// TIA Portal V19 export
FUNCTION "CallSettings" : Void   // FC8, LAD
// Call of settings blocks
// stored: IsIECCheckEnabled true, SetENOAutomatically false
BEGIN

REGION Network 1: Set set PLC date and time
   // Change local date and time of the PLC
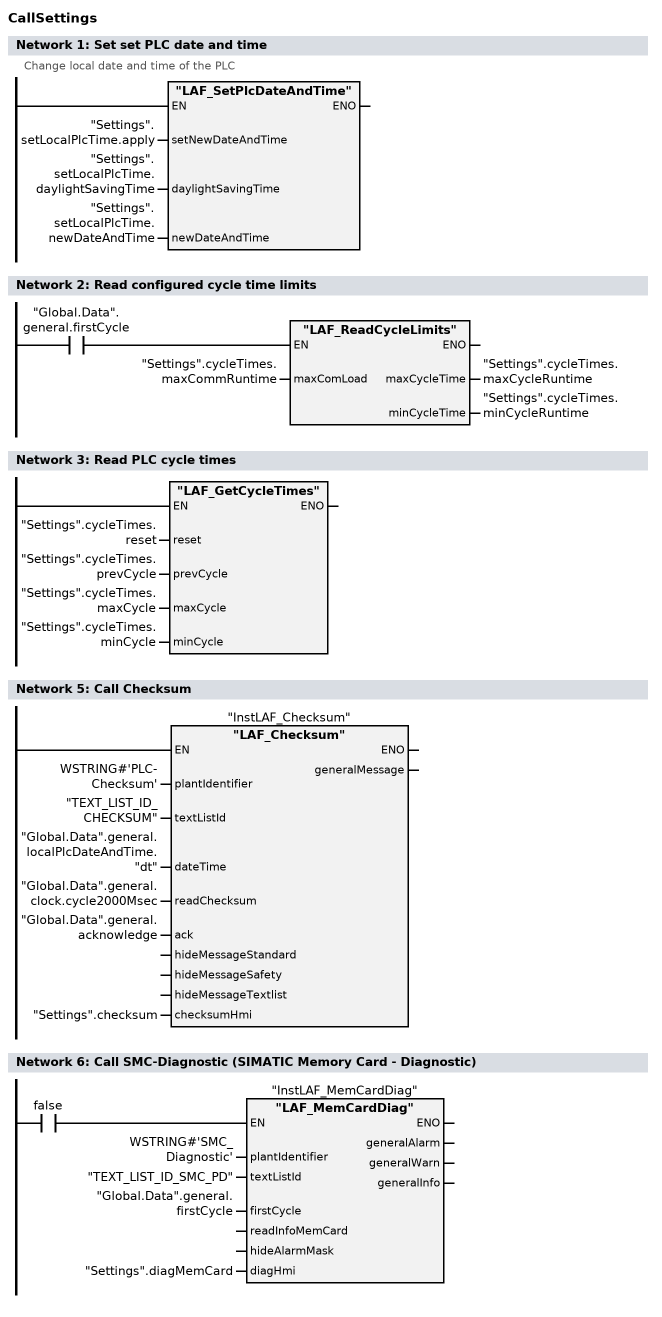
   RUNG wire#powerrail
      "LAF_SetPlcDateAndTime"(setNewDateAndTime := "Settings".setLocalPlcTime.apply, daylightSavingTime := "Settings".setLocalPlcTime.daylightSavingTime, newDateAndTime := "Settings".setLocalPlcTime.newDateAndTime)
   END_RUNG
   // the same network as SCL:
   "LAF_SetPlcDateAndTime"(setNewDateAndTime := "Settings".setLocalPlcTime.apply,
                           daylightSavingTime := "Settings".setLocalPlcTime.daylightSavingTime,
                           newDateAndTime := "Settings".setLocalPlcTime.newDateAndTime);
END_REGION

REGION Network 2: Read configured cycle time limits
   RUNG wire#powerrail
      Contact( "Global.Data".general.firstCycle )
      "LAF_ReadCycleLimits"(maxComLoad := "Settings".cycleTimes.maxCommRuntime, maxCycleTime => "Settings".cycleTimes.maxCycleRuntime, minCycleTime => "Settings".cycleTimes.minCycleRuntime)
   END_RUNG
   // the same network as SCL:
   IF "Global.Data".general.firstCycle THEN
       "LAF_ReadCycleLimits"(maxComLoad := "Settings".cycleTimes.maxCommRuntime,
                             maxCycleTime => "Settings".cycleTimes.maxCycleRuntime,
                             minCycleTime => "Settings".cycleTimes.minCycleRuntime);
   END_IF;
END_REGION

REGION Network 3: Read PLC cycle times
   RUNG wire#powerrail
      "LAF_GetCycleTimes"(reset := "Settings".cycleTimes.reset, prevCycle := "Settings".cycleTimes.prevCycle, maxCycle := "Settings".cycleTimes.maxCycle, minCycle := "Settings".cycleTimes.minCycle)
   END_RUNG
   // the same network as SCL:
   "LAF_GetCycleTimes"(reset := "Settings".cycleTimes.reset,
                       prevCycle := "Settings".cycleTimes.prevCycle,
                       maxCycle := "Settings".cycleTimes.maxCycle,
                       minCycle := "Settings".cycleTimes.minCycle);
END_REGION

REGION Network 4: Call PLC-Diagnostic
END_REGION

REGION Network 5: Call Checksum
   RUNG wire#powerrail
      "InstLAF_Checksum"(plantIdentifier := WSTRING#'PLC-Checksum', textListId := "TEXT_LIST_ID_CHECKSUM", dateTime := "Global.Data".general.localPlcDateAndTime."dt", readChecksum := "Global.Data".general.clock.cycle2000Msec, ack := "Global.Data".general.acknowledge, hideMessageStandard :=, hideMessageSafety :=, hideMessageTextlist :=, checksumHmi := "Settings".checksum, generalMessage =>)
   END_RUNG
   // the same network as SCL:
   "InstLAF_Checksum"(plantIdentifier := WSTRING#'PLC-Checksum',   // "LAF_Checksum"
                      textListId := "TEXT_LIST_ID_CHECKSUM",
                      dateTime := "Global.Data".general.localPlcDateAndTime."dt",
                      readChecksum := "Global.Data".general.clock.cycle2000Msec,
                      ack := "Global.Data".general.acknowledge,
                      checksumHmi := "Settings".checksum);
END_REGION

REGION Network 6: Call SMC-Diagnostic (SIMATIC Memory Card - Diagnostic)
   RUNG wire#powerrail
      Contact( false )
      "InstLAF_MemCardDiag"(plantIdentifier := WSTRING#'SMC_Diagnostic', textListId := "TEXT_LIST_ID_SMC_PD", firstCycle := "Global.Data".general.firstCycle, readInfoMemCard :=, hideAlarmMask :=, diagHmi := "Settings".diagMemCard, generalAlarm =>, generalWarn =>, generalInfo =>)
   END_RUNG
   // the same network as SCL:
   IF false THEN
       "InstLAF_MemCardDiag"(plantIdentifier := WSTRING#'SMC_Diagnostic',   // "LAF_MemCardDiag"
                             textListId := "TEXT_LIST_ID_SMC_PD",
                             firstCycle := "Global.Data".general.firstCycle,
                             diagHmi := "Settings".diagMemCard);
   END_IF;
END_REGION
END_FUNCTION
